// TIA Portal V17 export
// export: Created 2022-07-28T18:02:50.1916118Z, ExportSetting None, DisplayName Totally Integrated Automation Portal, DisplayVersion V17, DisplayName TIA Portal Openness, DisplayVersion V17, DisplayName TIA Portal Teamcenter Gateway, DisplayVersion V17, DisplayName TIA Portal Version Control Interface, DisplayVersion V17, DisplayName TIA Portal Test Suite Advanced, DisplayVersion V17, DisplayName SINAMICS Startdrive Advanced, DisplayVersion V17, DisplayName SINAMICS DCC, DisplayVersion V17, DisplayName SINAMICS Startdrive G130, G150, S120, S150, SINAMICS MV, S210, DisplayVersion V17, DisplayName SINAMICS Startdrive G110M, G120, G120C, G120D, G120P, G115D, DisplayVersion V17, DisplayName STEP 7 Professional, DisplayVersion V17, DisplayName SIMATIC Energy Suite, DisplayVersion V17, DisplayName STEP 7 CFC, DisplayVersion V17, DisplayName STEP 7 Safety, DisplayVersion V17, DisplayName WinCC Advanced / Unified PC, DisplayVersion V17, DisplayName SIMATIC Visualization Architect, DisplayVersion V17
FUNCTION_BLOCK "Lib_FB_Pump_Inv352_Base"   // FB79, SCL
{ S7_Optimized_Access := 'TRUE' }
// stored: AutoNumber false, MemoryReserve 100, SetENOAutomatically false
   VAR_INPUT
      I_Initialization { ExternalAccessible := 'False'; ExternalVisible := 'False'; ExternalWritable := 'False'} : Bool := FALSE;   // 1 = Restart PLC is active (First scan)
      IR_CycleTime { ExternalAccessible := 'False'; ExternalVisible := 'False'; ExternalWritable := 'False'} : Real := 0.0;   // Time of last PLC cycle, sec
      II_Obj_ID { ExternalAccessible := 'False'; ExternalVisible := 'False'; ExternalWritable := 'False'} : Int := -1;   // Tech ID of object
      I_CmdGeneralReset { ExternalAccessible := 'False'; ExternalVisible := 'False'; ExternalWritable := 'False'} : Bool;   // 0 ⮥ 1 = Input general reset ERROR/Interlocks
      I_One_1s { ExternalAccessible := 'False'; ExternalVisible := 'False'; ExternalWritable := 'False'} : Bool;   // 1 = One cycle per one seccond pulse
      I_EnableHorn { ExternalAccessible := 'False'; ExternalVisible := 'False'; ExternalWritable := 'False'} : Bool := TRUE;   // 1 = Set horn out befor start element
      I_EstopLocal { ExternalAccessible := 'False'; ExternalVisible := 'False'; ExternalWritable := 'False'} : Bool := TRUE;   // 0 = Emergency stop from local button is active (button is pressed)
      I_EstopHMI { ExternalAccessible := 'False'; ExternalVisible := 'False'; ExternalWritable := 'False'} : Bool := TRUE;   // 0 = HMI/WinCC Emergency stop active
      I_SuppyBox_Ok { ExternalAccessible := 'False'; ExternalVisible := 'False'; ExternalWritable := 'False'} : Bool := TRUE;   // 1 = Release from supply box where exist object
      I_ELSS_On { ExternalAccessible := 'False'; ExternalVisible := 'False'; ExternalWritable := 'False'} : Bool := TRUE;   // 1 = Emergency Local safety switch ON / Repair switch (IF 0 -> fault)
      I_MP_Ok { ExternalAccessible := 'False'; ExternalVisible := 'False'; ExternalWritable := 'False'} : Bool := TRUE;   // 1 = motor available - input should be wired directly to the motors circuit breaker input // 0 = motor not available - motor is disabled an an error is triggered
      I_ThermoDefend { ExternalAccessible := 'False'; ExternalVisible := 'False'; ExternalWritable := 'False'} : Bool := TRUE;   // 1 = Thermo defences is Ok
      I_TripBus { ExternalAccessible := 'False'; ExternalVisible := 'False'; ExternalWritable := 'False'} : Bool;   // 1 = Break connection with inverter
      I_EnableForward { ExternalAccessible := 'False'; ExternalVisible := 'False'; ExternalWritable := 'False'} : Bool := TRUE;   // 1 = motor is allowed to run in the forward direction // 0 = locked - motor is not allowed to run in the forward direction
      I_EnableReverse { ExternalAccessible := 'False'; ExternalVisible := 'False'; ExternalWritable := 'False'} : Bool;   // 1 = motor is allowed to run in the reverse direction // 0 = locked - motor is not allowed to run in the reverse direction
      I_CmdAutoFromInputFB { ExternalAccessible := 'False'; ExternalVisible := 'False'; ExternalWritable := 'False'} : Bool;   // 1 = Команди AutoMode беруться із входу FB // 0 = Команди AutoMode беруться із масиву AutoArray
      I_CmdAutoForward { ExternalAccessible := 'False'; ExternalVisible := 'False'; ExternalWritable := 'False'} : Bool;   // (if IB_CmdAutoFromInputFB==1) 1 = In auto mode the motor to run in Forward direction until the forward interlock becomes false, or this input is set low"
      I_CmdAutoReverse { ExternalAccessible := 'False'; ExternalVisible := 'False'; ExternalWritable := 'False'} : Bool;   // (if IB_CmdAutoFromInputFB==1) 1 = In auto mode the motor to run in Reverse direction until the forward interlock becomes false, or this input is set low"
      IR_AutoSpeedSP { ExternalAccessible := 'False'; ExternalVisible := 'False'; ExternalWritable := 'False'} : Real;   // Speed setpoint for auto mode from input, %
      I_ManLocalModeActive { ExternalAccessible := 'False'; ExternalVisible := 'False'; ExternalWritable := 'False'} : Bool;   // Switching in external mode ManualLocal if PRM.ManLocalPirority=1(hight)
      "I_CmdManLocalForward/Open" { ExternalAccessible := 'False'; ExternalVisible := 'False'; ExternalWritable := 'False'} : Bool;   // 1 = In ManualLocal mode the motor to run in Forward direction until the forward interlock becomes false, or this input is set low
      "I_CmdManLocalReverse/Close" { ExternalAccessible := 'False'; ExternalVisible := 'False'; ExternalWritable := 'False'} : Bool;   // 1 = In ManualLocal mode the motor to run in Reverse direction until the forward interlock becomes false, or this input is set low
      IB_InterlocksForward_8 { ExternalAccessible := 'False'; ExternalVisible := 'False'; ExternalWritable := 'False'} : Byte;   // <>0 = Interlock active - One or more from 8 Interlocks active // 1bit <--> 1 Interlock
      IB_InterlocksReverse_8 { ExternalAccessible := 'False'; ExternalVisible := 'False'; ExternalWritable := 'False'} : Byte;   // <>0 = Interlock active - One or more from 8 Interlocks active // 1bit <--> 1 Interlock
      IW_ExternalError_16 { ExternalAccessible := 'False'; ExternalVisible := 'False'; ExternalWritable := 'False'} : Word;   // <>0 = External error active - One or more from 16 error active // 1bit <--> 1 error
      I_ExternalWarning { ExternalAccessible := 'False'; ExternalVisible := 'False'; ExternalWritable := 'False'} : Bool;   // 1 = External Warning
      I_Termistor_Ok { ExternalAccessible := 'False'; ExternalVisible := 'False'; ExternalWritable := 'False'} : Bool := TRUE;   // 1 = Termistor sensor of motor is Ok
      IR_TimeTripInverter { ExternalAccessible := 'False'; ExternalVisible := 'False'; ExternalWritable := 'False'} : Real := 15.0;   // Time befor inverter self start/stop trip was detect, sec
      IR_SP_SpeedMax { ExternalAccessible := 'False'; ExternalVisible := 'False'; ExternalWritable := 'False'} : Real := 100.0;   // Maximus speed setpoint, %
      IR_SP_SpeedMin { ExternalAccessible := 'False'; ExternalVisible := 'False'; ExternalWritable := 'False'} : Real := 15.0;   // Minimum speed setpoint, %
   END_VAR
   VAR_OUTPUT
      Q_CmdForward { ExternalAccessible := 'False'; ExternalVisible := 'False'; ExternalWritable := 'False'} : Bool;   // 1 = Motor commanded forward /Activation output / State transferred to physical output
      Q_CmdReverse { ExternalAccessible := 'False'; ExternalVisible := 'False'; ExternalWritable := 'False'} : Bool;   // 1 = Motor commanded reverse / Activation output / State transferred to physical output
      Q_CmdHorn { ExternalAccessible := 'False'; ExternalVisible := 'False'; ExternalWritable := 'False'} : Bool;   // 1= Horn active
      Q_Reset { ExternalAccessible := 'False'; ExternalVisible := 'False'; ExternalWritable := 'False'} : Bool;   // 1 = Reset faults
      Q_Error { ExternalAccessible := 'False'; ExternalVisible := 'False'; ExternalWritable := 'False'} : Bool;   // This output indicates whether theres an error/fault condition in the motor
      Q_Warning { ExternalAccessible := 'False'; ExternalVisible := 'False'; ExternalWritable := 'False'} : Bool;   // This output indicates whether theres an warning condition in the motor
      Q_Auto { ExternalAccessible := 'False'; ExternalVisible := 'False'; ExternalWritable := 'False'} : Bool;   // 1= Automatic operating mode active
      Q_ManLocal { ExternalAccessible := 'False'; ExternalVisible := 'False'; ExternalWritable := 'False'} : Bool;   // 1= ManualLocal operating mode active
      Q_Stoped { ExternalAccessible := 'False'; ExternalVisible := 'False'; ExternalWritable := 'False'} : Bool;   // 1= Motor Stoped
      Q_Run { ExternalAccessible := 'False'; ExternalVisible := 'False'; ExternalWritable := 'False'} : Bool;   // 1= Motor running
      Q_RunForward { ExternalAccessible := 'False'; ExternalVisible := 'False'; ExternalWritable := 'False'} : Bool;   // 1= Motor running forward
      Q_RunReverse { ExternalAccessible := 'False'; ExternalVisible := 'False'; ExternalWritable := 'False'} : Bool;   // 1= Motor running forward
      Q_DataErr { ExternalAccessible := 'False'; ExternalVisible := 'False'; ExternalWritable := 'False'} : Bool;   // 1 = Transfer data error occured (ObjDB -> temp, ect)
      QR_SpeedSetpoint { ExternalAccessible := 'False'; ExternalVisible := 'False'; ExternalWritable := 'False'} : Real;   // Setpoint speed, %
      QR_SpeedActual { ExternalAccessible := 'False'; ExternalVisible := 'False'; ExternalWritable := 'False'} : Real;   // Actual speed, %
      QR_CurrentActual { ExternalAccessible := 'False'; ExternalVisible := 'False'; ExternalWritable := 'False'} : Real;   // Actual current, %
   END_VAR
   VAR_IN_OUT
      IQ_PLC_CycleInfo : Variant;   // Ref to data about PLC cycle
   END_VAR
   VAR
      s_RequestForward { ExternalAccessible := 'False'; ExternalVisible := 'False'; ExternalWritable := 'False'} : Bool;   // 1 = Request for start in forward dirrection for all modes
      s_RequestReverse { ExternalAccessible := 'False'; ExternalVisible := 'False'; ExternalWritable := 'False'} : Bool;   // 1 = Request for start in reverse dirrection for all modes
      s_Stopdown { ExternalAccessible := 'False'; ExternalVisible := 'False'; ExternalWritable := 'False'} : Bool;   // 1 = Stopdown is active
      s_EdgeAuto { ExternalAccessible := 'False'; ExternalVisible := 'False'; ExternalWritable := 'False'} : "Lib_FB_Edge";
      s_EdgeSim { ExternalAccessible := 'False'; ExternalVisible := 'False'; ExternalWritable := 'False'} : "Lib_FB_Edge";
      s_EdgeLocal { ExternalAccessible := 'False'; ExternalVisible := 'False'; ExternalWritable := 'False'} : "Lib_FB_Edge";
      s_EdgeError { ExternalAccessible := 'False'; ExternalVisible := 'False'; ExternalWritable := 'False'} : "Lib_FB_Edge";
      s_EdgeWarning { ExternalAccessible := 'False'; ExternalVisible := 'False'; ExternalWritable := 'False'} : "Lib_FB_Edge";
      s_EdgeActivForward { ExternalAccessible := 'False'; ExternalVisible := 'False'; ExternalWritable := 'False'} : "Lib_FB_Edge";
      s_EdgeActivRevers { ExternalAccessible := 'False'; ExternalVisible := 'False'; ExternalWritable := 'False'} : "Lib_FB_Edge";
   END_VAR
   VAR RETAIN
      s_Simulation { ExternalAccessible := 'False'; ExternalVisible := 'False'; ExternalWritable := 'False'} : Struct   // Data for simulation process
         Obj_DATA_BACKUP : Struct   // MOTOR NORMAL MODE DATA BACKUP FOR SIMULATION MODE
            Config : "_Pump_Inv352_Base_Config";
            Counters : "_Pump_Inv352_Base_Counters";
            sud_MotoHours_Electro : "_MotoHours_One";
            sud_MotoHours_Mech : "_MotoHours_One";
         END_STRUCT;
      END_STRUCT;
      s_Obj_Retain_BUp { ExternalAccessible := 'False'; ExternalVisible := 'False'; ExternalWritable := 'False'} : Struct
         Config : "_Pump_Inv352_Base_Config";
         Counters : "_Pump_Inv352_Base_Counters";
         Mode : "UDT_Mode";
      END_STRUCT;
   END_VAR
   VAR
      s_Moto { ExternalAccessible := 'False'; ExternalVisible := 'False'; ExternalWritable := 'False'} : "Lib_FB_MotSimp";
      s_TON_Horn { ExternalAccessible := 'False'; ExternalVisible := 'False'; ExternalWritable := 'False'} : "Lib_FB_Timer_ON_Simple";
      s_TON_AutoStartForward { ExternalAccessible := 'False'; ExternalVisible := 'False'; ExternalWritable := 'False'} : "Lib_FB_Timer_ON_Simple";
      s_TOF_AutoStopForward { ExternalAccessible := 'False'; ExternalVisible := 'False'; ExternalWritable := 'False'} : "Lib_FB_Timer_OFF_Simple";
      s_TON_AutoStartReverse { ExternalAccessible := 'False'; ExternalVisible := 'False'; ExternalWritable := 'False'} : "Lib_FB_Timer_ON_Simple";
      s_TOF_AutoStopReverse { ExternalAccessible := 'False'; ExternalVisible := 'False'; ExternalWritable := 'False'} : "Lib_FB_Timer_OFF_Simple";
      s_TP_ResetOut { ExternalAccessible := 'False'; ExternalVisible := 'False'; ExternalWritable := 'False'} : "Lib_FB_Timer_TP_Simple";
   END_VAR
   VAR_TEMP
      t_DataErr : Bool;   // 1 = Transfer data error occured (ObjDB -> temp, ect)
      t_ReleaseStart : Bool;   // 1 = Release for start in any mode
      t_RequestActive : Bool;   // 1 = Request is active for any mode in any dirrection
      t_RequestForwardActive : Bool;   // 1 = Request is active for any mode in forward dirrection
      t_RequestReverseActive : Bool;   // 1 = Request is active for any mode in reverse dirrection
      t_Startup : Bool;   // 1 = Startup of motor is active
      t_ResetLogic : Bool;   // 1 = Reset all signals for logic
      t_HornCompleted : Bool;   // 1 = Delay for horn was comleted
      ti_CMDLogic : Int;   // Command word for logic
      ti_NumObjDB : UInt;   // Number of DB for storage object data
      t_MaxObjects : UInt;   // Max number of objects in plant
      tr_HornTime : Real;   // Time for horn play, sec
      tr_SpeedSP_Logic : Real;   // Speed setpoint for logic, %
      t_ObjAny_HMI : DB_ANY;   // Ref to object data
      t_ObjVar_HMI : Variant;   // Ref to object data
      t_ObjAny_PLC : DB_ANY;   // Ref to object data
      t_ObjVar_PLC : Variant;   // Ref to object data
      t_ObjAny_Inv : DB_ANY;   // Ref to object data
      t_ObjVar_Inv : Variant;   // Ref to object data
      t_PB_HMI : Struct   // Buttons from HMI
         ResetError : Bool;   // + set-->CMD_ALMACK_tag -Reset errors pushbutton
         ManStop : Bool;   // - Stop in manual mode pushbutto
         ManRunForward : Bool;   // - Move forward in manual mode pushbutton
         ManRunReverse : Bool;   // - Move Reverse in manual mode pushbutton
         ResetInterlock : Bool;   // - Reset Interlock / Розблокувати
         ResetGeneralReset : Bool;   // -Reset Error + Interlock
         CntResetALL : Bool;   // - обнулити всі лічильники - (Total+Last)
         CntResetTimeTOT : Bool;   // - обнулити лічильник мотогодин (Total+Last)
         CntResetActTOT : Bool;   // - обнулити запусків (Total+Last)
         spare9 : Bool;
         spare10 : Bool;
         spare11 : Bool;
         spare12 : Bool;
         spare13 : Bool;
         spare14 : Bool;
         spare15 : Bool;
         spare16 : Bool;
         spare17 : Bool;
         spare18 : Bool;
         spare19 : Bool;
         spare20 : Bool;
         spare21 : Bool;
         spare22 : Bool;
         spare23 : Bool;
         spare24 : Bool;
         spare25 : Bool;
         spare26 : Bool;
         spare27 : Bool;
         spare28 : Bool;
         spare29 : Bool;
         spare30 : Bool;
         spare31 : Bool;
      END_STRUCT;
      t_Obj_HMI : "Lib_UDT_Pump_Inv352_Base_HMI";   // Object data
      t_Obj_PLC : "Lib_UDT_Pump_Inv352_Base_PLC";   // Object data
      t_Obj_Inv : "Lib_UDT_Inverter_352Tel";   // Object data
      t_PLC_CycleInfo : "Lib_PLC_CycleInfo";   // Data about PLC cycle
      t_AutoControl : "Lib_UDT_AutoControl";   // Data for auto control module for current element
      t_InternalData : "Lib_UDT_Int";   // Internal data
      t_AutoControl_CMD : Struct   // Commands from auto control module for current element
         CmdAutoForward : Bool;
         CmdAutoReverse : Bool;
         CmdAutoForwardRaw : Bool;
         CmdAutoReverseRaw : Bool;
      END_STRUCT;
      t_Buffer : Array[0..100] of Byte;   // Buffer for use serialize
      tui_DB_ShiftHMI : UInt;   // Object DB number shift
      tui_DB_ShiftPLC : UInt;   // Object DB number shift
      tui_DB_ShiftInv : UInt;
   END_VAR
BEGIN
   REGION Initialization/read data from out DB
       //Set internal data
       "Lib_FC_GenMoto_InitInternal"(#t_InternalData);

       //Reinit gen data
       #t_DataErr := false;
       #t_Obj_HMI.Config.w_enableExternalErrors_16 := w#16#FFFF;
       #t_Obj_HMI.Config.b_bypassInterlocksForward_8 := b#16#ff;
       #t_Obj_HMI.Config.b_bypassInterlocksReverse_8 := b#16#ff;
       #tr_HornTime := "D_General_ProgramDATA".r_HornTime;
       #t_MaxObjects := "D_General_ProgramDATA".ui_MaxObjects;
       #tui_DB_ShiftHMI := "D_General_ProgramDATA".ui_Shift_DB_HMI;
       #tui_DB_ShiftPLC := "D_General_ProgramDATA".ui_Shift_DB_PLC;
       #tui_DB_ShiftInv := "D_General_ProgramDATA".ui_Shift_DB_Bus;

       //Read data PLC
       VariantGet(SRC := #IQ_PLC_CycleInfo,
                  DST => #t_PLC_CycleInfo);

       //Read Object data
       //Reinit temp values
       #t_Obj_HMI := "D_ZeroTypes".Pump_Inv352_Base_HMI;
       #t_Obj_PLC := "D_ZeroTypes".Pump_Inv352_Base_PLC;
       #t_Obj_Inv := "D_ZeroTypes".Inverter_352Tel;

       IF #II_Obj_ID >= 0
       THEN
           //Read HMI data
           #ti_NumObjDB := INT_TO_UINT(#II_Obj_ID) + #tui_DB_ShiftHMI;
           #t_ObjAny_HMI := UINT_TO_DB_ANY(#ti_NumObjDB);
           #t_ObjVar_HMI := DB_ANY_TO_VARIANT(in := #t_ObjAny_HMI, err => #t_InternalData.i_Tmp);

           //If DB exist and convertion without error
           IF #t_InternalData.i_Tmp = 0
           THEN
               VariantGet(SRC := #t_ObjVar_HMI,
                          DST => #t_Obj_HMI);
           ELSE
               #t_DataErr := true;
           END_IF;

           //Read PLC data
           #ti_NumObjDB := INT_TO_UINT(#II_Obj_ID) + #tui_DB_ShiftPLC;
           #t_ObjAny_PLC := UINT_TO_DB_ANY(#ti_NumObjDB);
           #t_ObjVar_PLC := DB_ANY_TO_VARIANT(in := #t_ObjAny_PLC, err => #t_InternalData.i_Tmp);

           //If DB exist and convertion without error
           IF #t_InternalData.i_Tmp = 0
           THEN
               VariantGet(SRC := #t_ObjVar_PLC,
                          DST => #t_Obj_PLC);
           ELSE
               #t_DataErr := true;
           END_IF;

           //Read Inverter data
           #ti_NumObjDB := INT_TO_UINT(#II_Obj_ID) + #tui_DB_ShiftInv;
           #t_ObjAny_Inv := UINT_TO_DB_ANY(#ti_NumObjDB);
           #t_ObjVar_Inv := DB_ANY_TO_VARIANT(in := #t_ObjAny_Inv, err => #t_InternalData.i_Tmp);

           //If DB exist and convertion without error
           IF #t_InternalData.i_Tmp = 0
           THEN
               VariantGet(SRC := #t_ObjVar_Inv,
                          DST => #t_Obj_Inv);
           ELSE
               #t_DataErr := true;
           END_IF;

           //Check correct limits
           IF #IR_SP_SpeedMin > #IR_SP_SpeedMax
           THEN
               #t_DataErr := true;
           END_IF;
       ELSE
           #t_DataErr := true;
       END_IF;

       //Read general info data
       #t_AutoControl := "DB_AutoControl_arr".AutoControl_arr[#t_MaxObjects];
       CASE #II_Obj_ID OF
           0..999:  // ID of element in range
               #t_AutoControl := "DB_AutoControl_arr".AutoControl_arr[#II_Obj_ID];
           ELSE
               ;
       END_CASE;

       //Read retain data if initialization is active
       IF #I_Initialization
       THEN
           #t_Obj_HMI.Config := #s_Obj_Retain_BUp.Config;
           #t_Obj_HMI.Counters := #s_Obj_Retain_BUp.Counters;
           #t_Obj_PLC.Mode := #s_Obj_Retain_BUp.Mode;
       END_IF;
   END_REGION
   //---------------------------------------------------------------
   //---------------------------------------------------------------
   REGION Define CMD for block logic 
       //Reinit logic CMD
       #ti_CMDLogic := 0;

       "Lib_FC_GenMoto_ChoiceCMD"(I_Mode := #t_Obj_PLC.Mode,
                                  QI_CMD_Logic => #ti_CMDLogic,
                                  IQI_CMD_Global := #t_PLC_CycleInfo.CMD_GLOBAL,
                                  IQI_CMD_Auto := #t_AutoControl.Global_CMD,
                                  IQI_CMD_HMI := #t_Obj_HMI.i_CMD);

   END_REGION
   //---------------------------------------------------------------
   //---------------------------------------------------------------
   REGION Switch modes  
       "Lib_FC_GenMoto_SwitchMode"(I_ManLocalModeActive := #I_ManLocalModeActive,
                                   IQI_CMD_Logic := #ti_CMDLogic,
                                   IQ_Mode := #t_Obj_PLC.Mode,
                                   IQ_ObjDataConfig := #t_Obj_HMI.Config,
                                   IQ_BUpDataConfig := #s_Simulation.Obj_DATA_BACKUP.Config,
                                   IQ_ObjDataCounters := #t_Obj_HMI.Counters,
                                   IQ_BUpDataCounters := #s_Simulation.Obj_DATA_BACKUP.Counters);
   END_REGION
   //---------------------------------------------------------------
   //---------------------------------------------------------------
   REGION Commands & release for start in auto mode
       //Raw command for start in auto mode
       //-------------------------------------
       IF #I_CmdAutoFromInputFB
       THEN // Auto CMD from FB INPUT
           #t_AutoControl_CMD.CmdAutoForwardRaw := #I_CmdAutoForward;
           #t_AutoControl_CMD.CmdAutoReverseRaw := #I_CmdAutoReverse;
           #tr_SpeedSP_Logic := #IR_AutoSpeedSP;
       ELSE // Auto CMD from AutoControl_array DB
           #t_AutoControl_CMD.CmdAutoForwardRaw := (WORD_TO_UINT(#t_AutoControl.CTW.%W0) > 0);
           //AND #t_AutoControl.StatusGen.Release;
           #t_AutoControl_CMD.CmdAutoReverseRaw := (WORD_TO_UINT(#t_AutoControl.CTW.%W1) > 0);
           //AND #t_AutoControl.StatusGen.Release;
           #tr_SpeedSP_Logic := #t_AutoControl.SP_AutoMode;
       END_IF;
       //-------------------------------------
       //-------------------------------------
       //Processed auto mode commands
       #t_AutoControl_CMD.CmdAutoForward := #t_AutoControl_CMD.CmdAutoForwardRaw;//#s_TOF_AutoStopForward.QB_TimerOut;
       #t_AutoControl_CMD.CmdAutoReverse := #t_AutoControl_CMD.CmdAutoReverseRaw;//#s_TOF_AutoStopReverse.QB_TimerOut;

       //Reset release bit
       #t_AutoControl.StatusGen.Release := false;
   END_REGION
   //---------------------------------------------------------------
   //---------------------------------------------------------------
   REGION Convert commands to bit
       //Reinit all bits
       SCATTER(IN := #t_InternalData.d_Alw0,
               OUT => #t_PB_HMI);

       //Read commands and set apropriate bits
       CASE #ti_CMDLogic OF
           11:  //Stop in manual mode
               #t_PB_HMI.ManStop := true;
           12:  // Start forward dirrection in manual mode
               #t_PB_HMI.ManRunForward := true;
           13:  // Start reverse dirrection in manual mode
               #t_PB_HMI.ManRunReverse := true;
           31:  // Reset general (faults and interlocks)
               #t_PB_HMI.ResetGeneralReset := true;
           32: // Reset errors
               #t_PB_HMI.ResetError := true;
           33: //Reset interlocks
               #t_PB_HMI.ResetInterlock := true;
           40: //Reset all counters
               #t_PB_HMI.CntResetALL := true;
           41: //Reset counters of motohours
               #t_PB_HMI.CntResetTimeTOT := true;
           42: //Reset counters of starts
               #t_PB_HMI.CntResetActTOT := true;
           ELSE
               ;
       END_CASE;

       //General bits for logic
       //General reset
       #t_ResetLogic := #t_PB_HMI.ResetError
       OR #t_PB_HMI.ResetGeneralReset
       OR #I_CmdGeneralReset;

       //Reset for out of block
       #s_TP_ResetOut(IR_CycleTime := #IR_CycleTime,
                      IB_StartTimerInput := #t_ResetLogic,
                      IR_SpTime := 1.5);

   END_REGION
   //---------------------------------------------------------------
   //---------------------------------------------------------------
   REGION Proccess faults, warnings, interlocks and status bits

       REGION Reinit words
           // Reinit alarm words
           IF #t_ResetLogic
               OR #I_Initialization
               OR #t_Obj_PLC.Mode.Disable
               OR #t_Obj_PLC.Mode.Repair
           THEN
               #t_Obj_HMI.Status.w_ALW1 := #t_InternalData.w_Alw0;
               #t_Obj_HMI.Status.w_ALW2 := #t_InternalData.w_Alw0;
               #t_Obj_HMI.Status.w_ALW3 := #t_InternalData.w_Alw0;
               #t_Obj_HMI.Status.w_ALW4 := #t_InternalData.w_Alw0;
               #t_Obj_HMI.Status.w_ALW5 := #t_InternalData.w_Alw0;
               //#t_Obj_PLC.State := "DB_ZeroTypes".Motor_Inv352_WithoutSensors_PLC.State;
               #t_Obj_PLC.Alarm := "D_ZeroTypes".Pump_Inv352_Base_PLC.Alarm;
           END_IF;

           //Reinit STW words
           #t_Obj_HMI.Status.dw_STW_1 := #t_InternalData.d_Alw0;
           #t_Obj_HMI.Status.dw_STW_2 := #t_InternalData.d_Alw0;
           #t_Obj_HMI.Status.dw_STW := #t_InternalData.d_Alw0;

           //Reinit interlocks words
           #t_Obj_HMI.Status.dw_ILW_Frw := #t_InternalData.d_Alw0;
           #t_Obj_HMI.Status.dw_ILW_Rev := #t_InternalData.d_Alw0;
       END_REGION

       //Interlocks
       #t_Obj_PLC.Alarm.InterlockForward := ((#t_Obj_HMI.Config.b_bypassInterlocksForward_8
       AND #IB_InterlocksForward_8) <> b#16#0)
       AND NOT #t_Obj_PLC.Mode.Disable
       AND NOT #t_Obj_PLC.Mode.Service;

       #t_Obj_PLC.Alarm.InterlockReverse := ((#t_Obj_HMI.Config.b_bypassInterlocksReverse_8
       AND #IB_InterlocksReverse_8) <> b#16#0)
       AND NOT #t_Obj_PLC.Mode.Disable
       AND NOT #t_Obj_PLC.Mode.Service;

       #t_Obj_HMI.Status.dw_ILW_Frw.%B0 := #IB_InterlocksForward_8;
       #t_Obj_HMI.Status.dw_ILW_Rev.%B0 := #IB_InterlocksReverse_8;

       REGION Faults common for sim and gen modes
           IF NOT #t_Obj_PLC.Mode.Disable
           THEN
               //Emergency stop from HMI 
               #t_Obj_PLC.Alarm.EstopHMI := NOT #I_EstopHMI;

               //External warning
               #t_Obj_PLC.Alarm.ExtWarning := #I_ExternalWarning;

               //Internal warning 
               #t_Obj_PLC.Alarm.IntWarning := #t_Obj_PLC.Alarm.WarningInverter;

               //External error
               #t_Obj_HMI.Status.dw_EEW.%W0 := #IW_ExternalError_16;
               #t_Obj_PLC.Alarm.ExtError := (#IW_ExternalError_16
               AND #t_Obj_HMI.Config.w_enableExternalErrors_16) <> w#16#0;

               //Fault of supply box
               #t_Obj_PLC.Alarm.FaultSupplyBox := NOT #I_SuppyBox_Ok;

               //Both request
               #t_Obj_PLC.Alarm.BothCommandToStart := (#s_Moto.qs_Statuses.FltStartFwdBwdActive
               OR (NOT #t_ResetLogic
               AND #t_Obj_PLC.Alarm.BothCommandToStart))
               AND NOT #I_Initialization;
           END_IF;
       END_REGION

       REGION Faults different for gen and sim modes
           IF NOT #t_Obj_PLC.Mode.Simulation
               AND NOT #t_Obj_PLC.Mode.Disable
           THEN
               //Emergency stop from local 
               #t_Obj_PLC.Alarm.EstopLocal := (NOT #I_EstopLocal
               OR (NOT #t_ResetLogic
               AND #t_Obj_PLC.Alarm.EstopLocal))
               AND NOT #I_Initialization;

               //Local safety (repair) switch
               #t_Obj_PLC.Alarm.ELSS_Off := (NOT #I_ELSS_On
               OR (NOT #t_ResetLogic
               AND #t_Obj_PLC.Alarm.ELSS_Off))
               AND NOT #I_Initialization;

               //Motor circuit protection switch
               #t_Obj_PLC.Alarm.TripMP := (NOT #I_MP_Ok
               OR (NOT #t_ResetLogic
               AND #t_Obj_PLC.Alarm.TripMP))
               AND NOT #I_Initialization;

               //Unauthorized Start
               #t_Obj_PLC.Alarm.UnauthorizedStart := (#s_Moto.qs_Statuses.FltFwdContOff
               OR #s_Moto.qs_Statuses.FltRevContOff
               OR (NOT #t_ResetLogic
               AND #t_Obj_PLC.Alarm.UnauthorizedStart))
               AND NOT #I_Initialization;

               //Unauthorized Stop
               #t_Obj_PLC.Alarm.UnauthorizedStop := (#s_Moto.qs_Statuses.FltFwdContOn
               OR #s_Moto.qs_Statuses.FltRevContOn
               OR (NOT #t_ResetLogic
               AND #t_Obj_PLC.Alarm.UnauthorizedStop))
               AND NOT #I_Initialization;

               //Motor termistor
               #t_Obj_PLC.Alarm.TripTermistor := (NOT #I_Termistor_Ok
               OR (NOT #t_ResetLogic
               AND #t_Obj_PLC.Alarm.TripTermistor))
               AND NOT #I_Initialization;

               //Thermo defences
               #t_Obj_PLC.Alarm.TripThermoDefend := (NOT #I_ThermoDefend
               OR (NOT #t_ResetLogic
               AND #t_Obj_PLC.Alarm.TripThermoDefend))
               AND NOT #I_Initialization;

               //Inverter fault
               #t_Obj_PLC.Alarm.TripInverter := #t_Obj_Inv.Receive.STW.FaultActive
               OR #t_Obj_Inv.Receive.STW.LockoutActive;

               //Inverter warning
               #t_Obj_PLC.Alarm.WarningInverter := #t_Obj_Inv.Receive.STW.AlarmActive;

               //Trip connection with inverter
               #t_Obj_PLC.Alarm.TripBus := #I_TripBus;

               //Plausible error
               #t_Obj_PLC.Alarm.ErrPlausible := ((#s_RequestForward
               AND #s_Moto.qs_Statuses.RunRev)
               OR (#s_RequestReverse
               AND #s_Moto.qs_Statuses.RunFwd)
               OR (NOT #t_ResetLogic
               AND #t_Obj_PLC.Alarm.ErrPlausible))
               AND NOT #I_Initialization;

           ELSIF #t_Obj_PLC.Mode.Simulation
               AND NOT #t_Obj_PLC.Mode.Disable
           THEN

               CASE #ti_CMDLogic OF
                   100:  //Local emergency stop
                       #t_Obj_PLC.Alarm.EstopLocal := NOT #t_Obj_PLC.Alarm.EstopLocal;
                   101:  //Local repair switch
                       #t_Obj_PLC.Alarm.ELSS_Off := NOT #t_Obj_PLC.Alarm.ELSS_Off;
                   102:  //Motor protection
                       #t_Obj_PLC.Alarm.TripMP := NOT #t_Obj_PLC.Alarm.TripMP;
                   103:  //Brake fault
                       #t_Obj_PLC.Alarm.TripBrake := NOT #t_Obj_PLC.Alarm.TripBrake;
                   104:  //Self starting
                       #t_Obj_PLC.Alarm.UnauthorizedStart := NOT #t_Obj_PLC.Alarm.UnauthorizedStart;
                   105:  //Self stopping
                       #t_Obj_PLC.Alarm.UnauthorizedStop := NOT #t_Obj_PLC.Alarm.UnauthorizedStop;
                   106:  //Motor termistor
                       #t_Obj_PLC.Alarm.TripTermistor := NOT #t_Obj_PLC.Alarm.TripTermistor;
                   107:  //Circuit protection of brake
                       #t_Obj_PLC.Alarm.TripBrake_CP := NOT #t_Obj_PLC.Alarm.TripBrake_CP;
                   108:  //Cooling fault
                       #t_Obj_PLC.Alarm.TripCooling := NOT #t_Obj_PLC.Alarm.TripCooling;
                   109:  //Circuit protection of cooling
                       #t_Obj_PLC.Alarm.TripCooling_CP := NOT #t_Obj_PLC.Alarm.TripCooling_CP;
                   110:  //General fault of main drive
                       #t_Obj_PLC.Alarm.TripKMLine := NOT #t_Obj_PLC.Alarm.TripKMLine;
                   113:  //Both commands to motor is active
                       #t_Obj_PLC.Alarm.BothCommandToStart := NOT #t_Obj_PLC.Alarm.BothCommandToStart;
                   116:  //Thermo defences
                       #t_Obj_PLC.Alarm.TripThermoDefend := NOT #t_Obj_PLC.Alarm.TripThermoDefend;
                   117:  //Inverter fault
                       #t_Obj_PLC.Alarm.TripInverter := NOT #t_Obj_PLC.Alarm.TripInverter;
                   118: //Inverter warning
                       #t_Obj_PLC.Alarm.WarningInverter := NOT #t_Obj_PLC.Alarm.WarningInverter;
                   119: //Trip connection with inverter
                       #t_Obj_PLC.Alarm.TripBus := NOT #t_Obj_PLC.Alarm.TripBus;
                   120: //Plausible error
                       #t_Obj_PLC.Alarm.ErrPlausible := NOT #t_Obj_PLC.Alarm.ErrPlausible;
                   ELSE
                       ;
               END_CASE;

           END_IF;

           REGION Timers, edges ect.

           END_REGION

       END_REGION

       REGION Some faults is active

           #t_Obj_PLC.State.Error := #t_Obj_PLC.Alarm.EstopLocal
           OR #t_Obj_PLC.Alarm.EstopHMI
           OR #t_Obj_PLC.Alarm.ExtError
           OR #t_Obj_PLC.Alarm.FaultSupplyBox
           OR #t_Obj_PLC.Alarm.ELSS_Off
           OR #t_Obj_PLC.Alarm.TripMP
           OR #t_Obj_PLC.Alarm.TripBrake
           OR #t_Obj_PLC.Alarm.UnauthorizedStart
           OR #t_Obj_PLC.Alarm.UnauthorizedStop
           OR #t_Obj_PLC.Alarm.BothCommandToStart
           OR #t_Obj_PLC.Alarm.ErrPlausible
           OR #t_Obj_PLC.Alarm.TripTermistor
           OR #t_Obj_PLC.Alarm.TripBrake_CP
           OR #t_Obj_PLC.Alarm.TripCooling
           OR #t_Obj_PLC.Alarm.TripCooling_CP
           OR #t_Obj_PLC.Alarm.TripKMLine
           OR #t_Obj_PLC.Alarm.TripInverter;

       END_REGION
   END_REGION
   //---------------------------------------------------------------
   //---------------------------------------------------------------
   REGION Release for start in any mode
       #t_ReleaseStart := NOT #t_Obj_PLC.State.Error
       AND NOT #s_Moto.q_Fault
       AND NOT #t_Obj_PLC.Mode.Disable
       AND NOT #t_Obj_PLC.Mode.Repair
       AND NOT #s_Moto.qs_Statuses.AfterStpBlck
       AND NOT #s_EdgeAuto.QB_EdgeNeg
       AND NOT #s_EdgeSim.QB_EdgeNeg
       AND NOT #s_EdgeLocal.QB_EdgeNeg
       AND NOT #s_Stopdown
       AND NOT #I_Initialization;
   END_REGION
   //---------------------------------------------------------------
   //---------------------------------------------------------------
   REGION Requests for start in any dirrections
       REGION Request in forward dirrection
           //Release for start
           #s_RequestForward := #t_ReleaseStart
           AND NOT #t_Obj_PLC.Alarm.InterlockForward
           AND #I_EnableForward
           AND NOT #s_RequestReverse
           AND NOT #s_Moto.qs_Statuses.RunRev

           //Start command in auto mode
           AND ((#t_Obj_PLC.Mode.Auto
           AND #t_AutoControl_CMD.CmdAutoForward)

           //Start in manual remote mode
           OR ((#t_Obj_PLC.Mode.ManualRemote
           OR #t_Obj_PLC.Mode.Service)
           AND (#t_PB_HMI.ManRunForward
           OR #s_RequestForward)
           AND NOT #t_PB_HMI.ManStop)

           //Start in manual local mode
           OR (#t_Obj_PLC.Mode.ManualLocal
           AND #"I_CmdManLocalForward/Open")
           );
       END_REGION
       //---------------------------------------------------------------
       //---------------------------------------------------------------
       REGION Request in reverse dirrection
           //Release for start
           #s_RequestReverse := #t_ReleaseStart
           AND NOT #t_Obj_PLC.Alarm.InterlockReverse
           AND #I_EnableReverse
           AND NOT #s_RequestForward
           AND NOT #s_Moto.qs_Statuses.RunFwd

           //Start command in auto mode
           AND ((#t_Obj_PLC.Mode.Auto
           AND #t_AutoControl_CMD.CmdAutoReverse)

           //Start in manual remote mode
           OR ((#t_Obj_PLC.Mode.ManualRemote
           OR #t_Obj_PLC.Mode.Service)
           AND (#t_PB_HMI.ManRunReverse
           OR #s_RequestReverse)
           AND NOT #t_PB_HMI.ManStop)

           //Start in manual local mode
           OR (#t_Obj_PLC.Mode.ManualLocal
           AND #"I_CmdManLocalReverse/Close")
           );
       END_REGION
       //---------------------------------------------------------------
       //---------------------------------------------------------------
       REGION Logic for stopdown & startup bits 
           //Logic for stopdown bit 
           #s_Stopdown := NOT #s_RequestForward
           AND NOT #s_RequestReverse
           AND #s_Moto.qs_Statuses.Run;

           //Logic for startup bit
           #t_Startup := (#s_RequestForward
           OR #s_RequestReverse)
           AND NOT #s_Moto.qs_Statuses.Run;
       END_REGION

   END_REGION
   //---------------------------------------------------------------
   //---------------------------------------------------------------
   REGION Delays befor start motor; work with brake and cooling
       //Requests delay for auto mode
       //Timers TON for process auto mode commands
       //-------------------------------------
       #s_TON_AutoStartForward(IR_CycleTime := #IR_CycleTime,
                               IB_StartTimerInput := #s_RequestForward,
                               IB_ResetTimer := (NOT #t_Obj_PLC.State.Ready
                               AND NOT #s_Moto.qs_Statuses.Run)
                               OR NOT #t_Obj_PLC.Mode.Auto,
                               IR_SpTime := #t_Obj_HMI.Config.r_spTimeOnDelAuto);

       #s_TON_AutoStartReverse(IR_CycleTime := #IR_CycleTime,
                               IB_StartTimerInput := #s_RequestReverse,
                               IB_ResetTimer := (NOT #t_Obj_PLC.State.Ready
                               AND NOT #s_Moto.qs_Statuses.Run)
                               OR NOT #t_Obj_PLC.Mode.Auto,
                               IR_SpTime := #t_Obj_HMI.Config.r_spTimeOnDelAuto);

       //Process requests in any modes
       #t_RequestForwardActive := (NOT #t_Obj_PLC.Mode.Auto
       AND #s_RequestForward)
       OR (#t_Obj_PLC.Mode.Auto
       AND (#s_TOF_AutoStopForward.QB_TimerOut
       OR #s_TON_AutoStartForward.QB_TimerOut));

       #t_RequestReverseActive := (NOT #t_Obj_PLC.Mode.Auto
       AND #s_RequestReverse)
       OR (#t_Obj_PLC.Mode.Auto
       AND (#s_TOF_AutoStopReverse.QB_TimerOut
       OR #s_TON_AutoStartReverse.QB_TimerOut));

       #t_RequestActive := #t_RequestForwardActive
       OR #t_RequestReverseActive;

       //Horn delay
       //Timer for detect that horn is done
       #s_TON_Horn(IR_CycleTime := #IR_CycleTime,
                   IB_StartTimerInput := #t_RequestActive
                   AND #I_EnableHorn,
                   IB_ResetTimer := NOT #t_Obj_PLC.State.Ready
                   AND NOT #s_Moto.qs_Statuses.Run,
                   IR_SpTime := #tr_HornTime);

       #t_HornCompleted := (#I_EnableHorn
       AND #s_TON_Horn.QB_TimerOut)
       OR (NOT #I_EnableHorn
       AND #t_RequestActive);

       //Timers TOF for process auto mode commands
       //-------------------------------------
       #s_TOF_AutoStopForward(IR_CycleTime := #IR_CycleTime,
                              IB_StartTimerInput := #s_TON_AutoStartForward.QB_TimerOut
                              AND #t_HornCompleted,
                              IB_ResetTimer := (NOT #t_Obj_PLC.State.Ready
                              AND NOT #s_Moto.qs_Statuses.Run)
                              OR NOT #t_Obj_PLC.Mode.Auto,
                              IR_SpTime := #t_Obj_HMI.Config.r_spTimeOffDelAuto);

       #s_TOF_AutoStopReverse(IR_CycleTime := #IR_CycleTime,
                              IB_StartTimerInput := #s_TON_AutoStartReverse.QB_TimerOut
                              AND #t_HornCompleted,
                              IB_ResetTimer := (NOT #t_Obj_PLC.State.Ready
                              AND NOT #s_Moto.qs_Statuses.Run)
                              OR NOT #t_Obj_PLC.Mode.Auto,
                              IR_SpTime := #t_Obj_HMI.Config.r_spTimeOffDelAuto);


   END_REGION
   //---------------------------------------------------------------
   //---------------------------------------------------------------
   REGION Call block of motor 
       #s_Moto(i_StartFwd := #t_RequestForwardActive
               AND #t_HornCompleted,
               i_StartRev := #t_RequestReverseActive
               AND #t_HornCompleted,
               i_FdbckFwd := #t_Obj_Inv.Receive.RunningForward,
               i_FdbckRev := #t_Obj_Inv.Receive.RunningReverse,
               i_RestartingPLC := #I_Initialization,
               i_SimMode := #t_Obj_PLC.Mode.Simulation,
               ir_TimeCycle := #IR_CycleTime,
               ir_SPTimeFdbck := #IR_TimeTripInverter,
               ir_SPTimeRev := #t_Obj_HMI.Config.r_spTimeOffDir,
               ir_SPTimeNxtStrt := #t_Obj_HMI.Config.r_spTimeRestart);

       REGION Pulses for motor running
           #s_EdgeActivForward(IB_Initialisation := #I_Initialization,
                               IB_Input := #s_Moto.qs_Statuses.RunFwd
           );
           #s_EdgeActivRevers(IB_Initialisation := #I_Initialization,
                              IB_Input := #s_Moto.qs_Statuses.RunRev
           );
       END_REGION
   END_REGION
   //---------------------------------------------------------------
   //---------------------------------------------------------------
   REGION Define speed setpoint for logic & actual speed for simulation
       IF #t_RequestActive
           //OR #s_Moto.os_Statuses.Run
       THEN
           IF #t_Obj_PLC.Mode.Auto
           THEN
               IF #I_CmdAutoFromInputFB
               THEN // Auto CMD from FB INPUT
                   #tr_SpeedSP_Logic := #IR_AutoSpeedSP;
               ELSE // Auto CMD from AutoControl_array DB
                   #tr_SpeedSP_Logic := #t_AutoControl.SP_AutoMode;
               END_IF;
           ELSE
               #tr_SpeedSP_Logic := #t_Obj_HMI.Config.r_spSpeed;
           END_IF;

           //Chech setpoint limits
           IF #tr_SpeedSP_Logic > #IR_SP_SpeedMax
           THEN
               #tr_SpeedSP_Logic := #IR_SP_SpeedMax;
           END_IF;

           IF #tr_SpeedSP_Logic < #IR_SP_SpeedMin
           THEN
               #tr_SpeedSP_Logic := #IR_SP_SpeedMin;
           END_IF;
       ELSE
           #tr_SpeedSP_Logic := 0.0;
       END_IF;

       //Define actual value of speed for simulation mode as set speed
       IF #t_Obj_PLC.Mode.Simulation
       THEN
           #t_Obj_Inv.Receive.r_ActualSpeed := #tr_SpeedSP_Logic;
       END_IF;
   END_REGION
   //---------------------------------------------------------------
   //---------------------------------------------------------------
   REGION Counters
       //Maintenance counters
       "Lib_FC_General_CountMotoHours"(II_Obj_ID := #II_Obj_ID,
                                       I_One_1s := #I_One_1s,
                                       I_Run := #s_Moto.qs_Statuses.Run,
                                       I_PosPulseSimMode := #s_EdgeSim.QB_EdgePos,
                                       I_NegPulseSimMode := #s_EdgeSim.QB_EdgeNeg,
                                       Q_MaintenanceElectroServ => #t_Obj_PLC.Alarm.MaintenanceElectroServ,
                                       Q_MaintenanceMechanoServ => #t_Obj_PLC.Alarm.MaintenanceMechanoServ,
                                       IQUD_BacUpElectro := #s_Simulation.Obj_DATA_BACKUP.sud_MotoHours_Electro,
                                       IQUD_BacUpMechanic := #s_Simulation.Obj_DATA_BACKUP.sud_MotoHours_Mech);

       //Total operating time
       IF #s_Moto.qs_Statuses.Run
           AND #I_One_1s
       THEN
           #t_Obj_HMI.Counters.di_TimeOper_Tot += 1;
       END_IF;

       //Counter starts
       IF #s_EdgeActivForward.QB_EdgePos
           OR #s_EdgeActivRevers.QB_EdgePos
       THEN
           #t_Obj_HMI.Counters.di_Activ_tot += 1;
       END_IF;

       //Reset general counters
       IF #t_PB_HMI.CntResetALL
       THEN
           #t_Obj_HMI.Counters.di_TimeOper_Tot := 0;
           #t_Obj_HMI.Counters.di_Activ_tot := 0;
       END_IF;

       IF #t_PB_HMI.CntResetTimeTOT
       THEN
           #t_Obj_HMI.Counters.di_TimeOper_Tot := 0;
       END_IF;

       IF #t_PB_HMI.CntResetActTOT
       THEN
           #t_Obj_HMI.Counters.di_Activ_tot := 0;
       END_IF;
   END_REGION
   //---------------------------------------------------------------
   //---------------------------------------------------------------
   REGION General states
       IF NOT #t_Obj_PLC.Mode.Disable
           AND NOT #t_Obj_PLC.Mode.Repair
       THEN
           //General states 
           #t_Obj_PLC.Alarm.ForwardEnable := #I_EnableForward;
           #t_Obj_PLC.Alarm.ReverseEnable := #I_EnableReverse;
           #t_Obj_PLC.Alarm.InCmdAutoForward := #t_AutoControl_CMD.CmdAutoForward;
           #t_Obj_PLC.Alarm.InCmdAutoReverse := #t_AutoControl_CMD.CmdAutoReverse;
           #t_Obj_PLC.Alarm.SigOutForward := #Q_CmdForward;
           #t_Obj_PLC.Alarm.SigOutReverse := #Q_CmdReverse;
           #t_Obj_PLC.Alarm.RequestForward := #s_RequestForward;
           #t_Obj_PLC.Alarm.RequestReverse := #s_RequestReverse;
           #t_Obj_PLC.Alarm.PauseStart := #s_Moto.qs_Statuses.AfterStpBlck;
           #t_Obj_PLC.Alarm.RunForward := #s_Moto.qs_Statuses.RunFwd;
           #t_Obj_PLC.Alarm.RunReverse := #s_Moto.qs_Statuses.RunRev;

           #t_Obj_PLC.State.Warning := #I_ExternalWarning
           OR #t_Obj_PLC.Alarm.IntWarning;
           #t_Obj_PLC.State.Maintenance := #t_Obj_PLC.Alarm.MaintenanceElectroServ
           OR #t_Obj_PLC.Alarm.MaintenanceMechanoServ;
           #t_Obj_PLC.State.Interlocked := #t_Obj_PLC.Alarm.InterlockForward
           OR #t_Obj_PLC.Alarm.InterlockReverse;
           #t_Obj_PLC.State.Ready := #t_ReleaseStart;
           #t_Obj_PLC.State.Stoped := NOT #s_Moto.qs_Statuses.Run
           AND NOT #s_Moto.qs_Statuses.AfterStpBlck;
           #t_Obj_PLC.State.Run := #s_Moto.qs_Statuses.Run;
           #t_Obj_PLC.State.RunForward := #s_Moto.qs_Statuses.RunFwd;
           #t_Obj_PLC.State.RunRevers := #s_Moto.qs_Statuses.RunRev;
           #t_Obj_PLC.State.Startup := (#s_RequestForward
           AND NOT #s_Moto.qs_Statuses.RunFwd)
           OR (#s_RequestReverse
           AND NOT #s_Moto.qs_Statuses.RunRev);
           #t_Obj_PLC.State.Shutdown := #s_Stopdown;
       END_IF;

       //States for all modes
       #t_Obj_PLC.Alarm.Disable := #t_Obj_PLC.Mode.Disable;
       #t_Obj_PLC.Alarm.ManualRemote := #t_Obj_PLC.Mode.ManualRemote;
       #t_Obj_PLC.Alarm.Auto := #t_Obj_PLC.Mode.Auto;
       #t_Obj_PLC.Alarm.ManualLocal := #t_Obj_PLC.Mode.ManualLocal;
       #t_Obj_PLC.Alarm.Service := #t_Obj_PLC.Mode.Service;
       #t_Obj_PLC.Alarm.RepairOn := #t_Obj_PLC.Mode.Repair;
       #t_Obj_PLC.Alarm.IndependentOn := #t_Obj_PLC.Mode.Independent;
       #t_Obj_PLC.Alarm.SimulationOn := #t_Obj_PLC.Mode.Simulation;
       #t_Obj_PLC.Alarm.RepairOff := NOT #t_Obj_PLC.Mode.Repair;
       #t_Obj_PLC.Alarm.IndependentOff := NOT #t_Obj_PLC.Mode.Independent;
       #t_Obj_PLC.Alarm.SimulationOff := NOT #t_Obj_PLC.Mode.Simulation;
       #t_Obj_PLC.Alarm.Stopped := NOT #s_Moto.qs_Statuses.Run;

       REGION Pulses for new states
           #s_EdgeError(IB_Initialisation := #I_Initialization,
                        IB_Input := #t_Obj_PLC.State.Error);
           #s_EdgeWarning(IB_Initialisation := #I_Initialization,
                          IB_Input := #t_Obj_PLC.State.Warning);
       END_REGION
   END_REGION
   //---------------------------------------------------------------
   //---------------------------------------------------------------
   REGION PLC states + Counter
       "Lib_FC_Mot_CycleInfo_Count_State"(Alarm := #t_Obj_PLC.State.Error,
                                          AlarmNew := #s_EdgeError.QB_EdgePos,
                                          Warning := #t_Obj_PLC.State.Warning,
                                          WarningNew := #s_EdgeWarning.QB_EdgePos,
                                          Estop := #t_Obj_PLC.Alarm.EstopLocal
                                          OR #t_Obj_PLC.Alarm.EstopHMI,
                                          Interlocked := #t_Obj_PLC.State.Interlocked,
                                          InterlockBypassed := false,
                                          Manual := #t_Obj_PLC.Mode.ManualRemote
                                          OR #t_Obj_PLC.Mode.ManualLocal,
                                          Simulation := #t_Obj_PLC.Mode.Simulation,
                                          Error_PSL := NOT #I_SuppyBox_Ok,
                                          PLC_CycleInfo := #t_PLC_CycleInfo);

   END_REGION
   //---------------------------------------------------------------
   //---------------------------------------------------------------
   REGION Write STW and Alarm bits into words

       //Wrapping Alarm bits in words
       #t_InternalData.di_Tmp := 0;
       #t_InternalData.i_Tmp := Serialize(SRC_VARIABLE := #t_Obj_PLC.Alarm, DEST_ARRAY => #t_Buffer, POS := #t_InternalData.di_Tmp);
       #t_Obj_HMI.Status.w_ALW1.%B0 := #t_Buffer[0];
       #t_Obj_HMI.Status.w_ALW1.%B1 := #t_Buffer[1];
       #t_Obj_HMI.Status.w_ALW2.%B0 := #t_Buffer[2];
       #t_Obj_HMI.Status.w_ALW2.%B1 := #t_Buffer[3];
       #t_Obj_HMI.Status.w_ALW3.%B0 := #t_Buffer[4];
       #t_Obj_HMI.Status.w_ALW3.%B1 := #t_Buffer[5];
       #t_Obj_HMI.Status.w_ALW4.%B0 := #t_Buffer[6];
       #t_Obj_HMI.Status.w_ALW4.%B1 := #t_Buffer[7];

       //Wrapping STW bits
       //States
       #t_InternalData.di_Tmp := 0;
       #t_InternalData.i_Tmp := Serialize(SRC_VARIABLE := #t_Obj_PLC.State, DEST_ARRAY => #t_Buffer, POS := #t_InternalData.di_Tmp);

       //Modes
       #t_InternalData.di_Tmp := 5;
       #t_InternalData.i_Tmp := Serialize(SRC_VARIABLE := #t_Obj_PLC.Mode, DEST_ARRAY => #t_Buffer, POS := #t_InternalData.di_Tmp);

       #t_Obj_HMI.Status.dw_STW.%B0 := #t_Buffer[0]; //States W1
       #t_Obj_HMI.Status.dw_STW.%B1 := #t_Buffer[1]; //States W2
       #t_Obj_HMI.Status.dw_STW.%B2 := #t_Buffer[2] OR #t_Buffer[5]; //Modes W1
       #t_Obj_HMI.Status.dw_STW.%B3 := #t_Buffer[6]; //Modes W2

   END_REGION
   //---------------------------------------------------------------
   //---------------------------------------------------------------
   REGION Write data to HMI and BUp storage
       //HMI data
       #t_Obj_HMI.i_ID := #II_Obj_ID;
       #t_Obj_HMI.i_CLSID := 77;
       #t_Obj_HMI.Status.w_FaultWord := #t_Obj_Inv.Receive.w_Fault;
       #t_Obj_HMI.Status.w_WarningWord := #t_Obj_Inv.Receive.w_Warning;
       #t_Obj_HMI.Status.r_ActualSpeed := #t_Obj_Inv.Receive.r_ActualSpeed;
       #t_Obj_HMI.Status.r_SetpointSpeed := #tr_SpeedSP_Logic;
       #t_Obj_HMI.Status.r_ActualCurrentPrc := #t_Obj_Inv.Receive.r_ActualCurrent;
       #t_Obj_HMI.Status.r_ActualTorque := #t_Obj_Inv.Receive.r_ActualTorque;
       IF #t_Obj_HMI.Config.r_spRefCurrent > 0.0
       THEN
           #t_Obj_HMI.Status.r_ActualCurrentAmp := #t_Obj_Inv.Receive.r_ActualCurrent/100.0 * #t_Obj_HMI.Config.r_spRefCurrent;
       ELSE
           #t_Obj_HMI.Status.r_ActualCurrentAmp := 0.0;
       END_IF;

       IF #t_Obj_HMI.Config.r_spRefFreq > 0.0
       THEN
           #t_Obj_HMI.Status.r_ActualFreq := #t_Obj_Inv.Receive.r_ActualSpeed / 100.0 * #t_Obj_HMI.Config.r_spRefFreq;
       ELSE
           #t_Obj_HMI.Status.r_ActualFreq := 0.0;
       END_IF;

       IF #t_Obj_HMI.Config.r_spRefRPM > 0.0
       THEN
           #t_Obj_HMI.Status.r_ActualRPM := #t_Obj_Inv.Receive.r_ActualSpeed / 100.0 * #t_Obj_HMI.Config.r_spRefRPM;
       ELSE
           #t_Obj_HMI.Status.r_ActualRPM := 0.0;
       END_IF;

       IF #t_Obj_HMI.Config.r_spRefPower > 0.0
       THEN
           #t_Obj_HMI.Status.r_ActualPower := 400.0 * #t_Obj_HMI.Status.r_ActualCurrentAmp / 1000.0;
       ELSE
           #t_Obj_HMI.Status.r_ActualPower := 0.0;
       END_IF;

       //BUp retain data
       //Read retain data if initialization is active
       IF NOT #I_Initialization
       THEN
           #s_Obj_Retain_BUp.Config := #t_Obj_HMI.Config;
           #s_Obj_Retain_BUp.Counters := #t_Obj_HMI.Counters;
           #s_Obj_Retain_BUp.Mode := #t_Obj_PLC.Mode;
       END_IF;
   END_REGION
   //---------------------------------------------------------------
   //---------------------------------------------------------------
   REGION Wrap data for automode module
       #t_AutoControl.STW_HMI := #t_InternalData.d_Alw0;
       #t_AutoControl.STW := #t_InternalData.d_Alw0;

       #t_AutoControl.Mode := #t_Obj_PLC.Mode;
       #t_AutoControl.CLSID := #t_Obj_HMI.i_CLSID;
       #t_AutoControl.StatusGen.Fault := #t_Obj_PLC.State.Error;
       #t_AutoControl.StatusGen.Ready := #t_Obj_PLC.State.Ready;
       #t_AutoControl.StatusGen.ControlAchieve := (#t_AutoControl_CMD.CmdAutoForward
       AND #s_Moto.qs_Statuses.RunFwd)
       OR (#t_AutoControl_CMD.CmdAutoReverse
       AND #s_Moto.qs_Statuses.RunRev);

       #t_InternalData.di_Tmp := 0;
       #t_InternalData.i_Tmp := Serialize(SRC_VARIABLE := #t_AutoControl.StatusGen, DEST_ARRAY => #t_Buffer, POS := #t_InternalData.di_Tmp);
       #t_InternalData.di_Tmp := 2;
       #t_InternalData.i_Tmp := Serialize(SRC_VARIABLE := #t_AutoControl.Mode, DEST_ARRAY => #t_Buffer, POS := #t_InternalData.di_Tmp);

       #t_AutoControl.STW_HMI.%B0 := #t_Buffer[0];
       #t_AutoControl.STW_HMI.%B1 := #t_Buffer[1];
       #t_AutoControl.STW_HMI.%B2 := #t_Buffer[2];
       #t_AutoControl.STW_HMI.%B3 := #t_Buffer[3];
       #t_AutoControl.STW_HMI.%X16 := false;

       IF #t_AutoControl_CMD.CmdAutoForward
           AND #s_Moto.qs_Statuses.RunFwd
       THEN
           #t_AutoControl.STW.%W0 := #t_AutoControl.CTW.%W0;
       END_IF;

       IF #t_AutoControl_CMD.CmdAutoReverse
           AND #s_Moto.qs_Statuses.RunRev
       THEN
           #t_AutoControl.STW.%W1 := #t_AutoControl.CTW.%W1;
       END_IF;
   END_REGION
   //---------------------------------------------------------------
   //---------------------------------------------------------------
   REGION Write data for inverter module
       #t_Obj_Inv.Send.r_SetpointSpeed := #tr_SpeedSP_Logic;

       #t_Obj_Inv.Send.CTW.OFF1 := (#s_Moto.q_CmdRunFwd
       OR #s_Moto.q_CmdRunRev);
       #t_Obj_Inv.Send.CTW.OFF2 := NOT #s_Stopdown;
       #t_Obj_Inv.Send.CTW.OFF3 := NOT #t_Obj_PLC.State.Error
       AND NOT #t_Obj_PLC.State.Interlocked
       AND NOT #t_Obj_PLC.Mode.Disable
       AND NOT #t_Obj_PLC.Mode.Simulation
       OR NOT #s_Moto.qs_Statuses.Run
       OR #s_TP_ResetOut.QB_TimerOut;
       #t_Obj_Inv.Send.CTW.Acknowlege := #s_TP_ResetOut.QB_TimerOut;
       #t_Obj_Inv.Send.CTW.ChangeDir := #s_Moto.q_CmdRunRev;

   END_REGION
   //---------------------------------------------------------------
   //---------------------------------------------------------------
   REGION Write data to out DB
       //Write data  PLC
       VariantPut(SRC := #t_PLC_CycleInfo,
                  DST := #IQ_PLC_CycleInfo);

       //Write Object data
       //DB num 
       IF #II_Obj_ID >= 0
           AND NOT #t_DataErr
       THEN
           //Write HMI data
           VariantPut(SRC := #t_Obj_HMI,
                      DST := #t_ObjVar_HMI);

           //Write PLC data
           VariantPut(SRC := #t_Obj_PLC,
                      DST := #t_ObjVar_PLC);

           //Write inverter data
           VariantPut(SRC := #t_Obj_Inv,
                      DST := #t_ObjVar_Inv);
       ELSE
           #t_DataErr := true;
       END_IF;

       //Write general info data
       CASE #II_Obj_ID OF
           0..999:  // ID of element in range
               "DB_AutoControl_arr".AutoControl_arr[#II_Obj_ID] := #t_AutoControl;
           ELSE
               ;
       END_CASE;

   END_REGION
   //---------------------------------------------------------------
   //---------------------------------------------------------------
   REGION Outputs of block
       #Q_CmdForward := #s_Moto.q_CmdRunFwd
       AND NOT #t_Obj_PLC.Mode.Simulation;
       #Q_CmdReverse := #s_Moto.q_CmdRunRev
       AND NOT #t_Obj_PLC.Mode.Simulation;
       #Q_CmdHorn := #I_EnableHorn
       AND NOT #t_HornCompleted
       AND (#s_RequestForward
       OR #s_RequestReverse)
       AND NOT #t_Obj_PLC.Mode.Simulation;
       #Q_Reset := #s_TP_ResetOut.QB_TimerOut;
       #Q_Error := #t_Obj_PLC.State.Error;
       #Q_Warning := #t_Obj_PLC.State.Warning;
       #Q_Auto := #t_Obj_PLC.Mode.Auto;
       #Q_ManLocal := #t_Obj_PLC.Mode.ManualLocal;
       #Q_Stoped := #t_Obj_PLC.State.Stoped;
       #Q_Run := #t_Obj_PLC.State.Run;
       #Q_RunForward := #t_Obj_PLC.State.RunForward;
       #Q_RunReverse := #t_Obj_PLC.State.RunRevers;
       #Q_DataErr := #t_DataErr;
       #QR_SpeedSetpoint := #t_Obj_Inv.Receive.r_ActualSpeed;
       #QR_SpeedActual := #tr_SpeedSP_Logic;
       #QR_CurrentActual := #t_Obj_Inv.Receive.r_ActualCurrent;
   END_REGION

   //Test text 17.02.2022
END_FUNCTION_BLOCK
